// TIA Portal V19 export
DATA_BLOCK "DB_Dosi_Overview"   // DB88
{ S7_Optimized_Access := 'FALSE' }
// stored: AutoNumber false
   VAR RETAIN
      LZ_Count : Array[1..13] of DWord;   // * erst DZ je 1 DW
      DP_Count : Array[1..40] of DWord;   // * dann DP je 2 DW (Auto/Hand)(Feldlänge := DZ + 2*DP)
   END_VAR
BEGIN
   LZ_Count[1..13] := 16#0000_0000;
   DP_Count[1..40] := 16#0000_0000;
END_DATA_BLOCK
